// TIA Portal V18 export
DATA_BLOCK "CheckPositioningOrder_IDB"   // DB3
VERSION : 0.1
// stored: AutoNumber true, DBAccessibleFromOPCUA true, DBAccessibleFromWebserver true, InstanceOfName CheckPositioningOrder, InstanceOfType FB
"CheckPositioningOrder"
   // VAR_INPUT
   //    "V90Servo[3]" : Struct
   //       i : Int;
   //       nError : Int;
   //       nWarning : Int;
   //       nPositionListNo : Int;
   //       Pos : "PosList";
   //       Point : Array[0..39] of Struct
   //          Start : Bool;
   //          Achieve : Bool;
   //       END_STRUCT;
   //    END_STRUCT;
   // END_VAR
   // VAR_OUTPUT
   //    HaveAxisStart : Bool;
   //    AxisStartNumber : Int;
   // END_VAR
   // VAR
   //    Index : Int;
   // END_VAR
BEGIN
END_DATA_BLOCK
